FUNCTION TryConvert_UINT_TO_UINT : BOOL
VAR_INPUT
	in : UINT;
	out : REFERENCE TO UINT;
END_VAR

out := in;
TryConvert_UINT_TO_UINT := TRUE;

END_FUNCTION

(* stored: Version 1.1.0.1, ProductVersion 3.1.4024.12
   POU TryConvert_UINT_TO_UINT: Id {0028009a-ad1f-4a91-b201-cb9fad8cea56}, SpecialFunc None *)
